VAR_GLOBAL
    KommAnVisu                 : INT;      (* Kommunikation an die Visualisierung *)
    KommVonVisu                : INT;      (* Kommunikation von der Visualisierung *)
    belegt                     : BOOL;     (* true = erzeugt Dummyteil, false = keine Auswirkungen (nur Handauflage) *)
    daten_gebucht              : BOOL;
    SteuerStatus               : DUT_Visu_SteuerStatus;

    // Frequenzumrichter
	Trans_Bandseite				: DUT_SEW_FU_Visu; 		//#Tab: 3520 Transport Bandseite #Name: Transport Bandseite X-Achse

    // Servoregler
	Y_Achse						: DUT_Achse_Service;	//#Tab: 3520 Transport Bandseite #Name: Y-Achse 
	X_Achse						: DUT_Achse_Service;	//#Tab: 3520 Transport Bandseite #Name: X-Achse Längsanschlag

    // Ventile
	 Laengsanschl        		: DUT_Ventil_VISU;      //#Tab: 3520 Transport Bandseite #Name: Bandseite Längsanschlag
	 Schienenklemm        		: DUT_Ventil_VISU;      //#Tab: 3520 Transport Bandseite #Name: Schienenklemmung

	refresh2					: BOOL;

END_VAR

VAR_GLOBAL PERSISTENT
    Schrittnummer           : INT;
    Kopfdaten               : DUT_Kopfdaten;
    Kopfdaten_default       : DUT_Kopfdaten;
    Jobdaten                : ARRAY[1..GVL_3000.cSize_Jobdaten] OF DUT_Jobdaten;
    Jobdaten_default        : ARRAY[1..GVL_3000.cSize_Jobdaten] OF DUT_Jobdaten;
	aktJob					: DUT_Jobdaten;
	iJobNr					: INT := 1;

    //para_Vorlage             : REAL := 0.0; //#Typ: VParam #Tab:  #Name:  #Einheit:mm #Min: 1 #Max: 100 #Format:F1
END_VAR

(* stored: Version 1.1.0.1
   GVL GVL_Visu_3520: Id {87d8f60e-845b-495e-b69f-fc19ba2f7ab3} *)
